FUNCTION_BLOCK bfb_peak
  (* Standard: 61499-2 *)
  (* Version 0.1, 2018-00-09, palme, DESKTOP-TGOEKBD *)
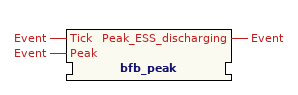
  EVENT_INPUT
    Tick;
    Peak;
  END_EVENT
  EVENT_OUTPUT
    Peak_ESS_discharging;
  END_EVENT
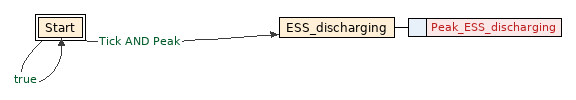
  EC_STATES
    Start;
    ESS_discharging : -> Peak_ESS_discharging;
  END_STATES
  EC_TRANSITIONS
    Start TO ESS_discharging := Tick AND Peak;
    Start TO Start := true;
  END_TRANSITIONS
END_FUNCTION_BLOCK
